Fanuc KAREL source: kt00224.KL

-- PROVISIONAL review KL for V1013-1; original PC SHA256 8b9f0a0df4764c2e2a0997e457185a337277f0c3b9f855f1c93c95c441e69a34
-- Incomplete behavior may be omitted. Consult companion uncertainty JSON. Do not deploy.
PROGRAM KT00224
%NOLOCKGROUP
VAR
  OUT : INTEGER
-- UNRESOLVED_DECL H1 type=002017
-- UNRESOLVED_DECL H2 type=002017
BEGIN
  -- UNRESOLVED_PC offsets 5-19; opcodes 2E,22,9D,33,B4
  -- UNRESOLVED_PC offsets 24-38; opcodes 2E,22,9D,33,B4
  -- UNRESOLVED_PC offsets 43-57; opcodes 2E,22,9D,33,B4
  -- UNRESOLVED_PC offsets 62-76; opcodes 2E,22,9D,33,B4
  -- UNRESOLVED_PC offsets 81-106; opcodes 22,9D,33,B3,22,9D,33,B3,46,23
  -- UNRESOLVED_PC offsets 111-115; opcodes 7F
END KT00224
